INTERFACE PUBLIC LogCore EXTENDS __SYSTEM.IQueryInterface

// Logger method.
// Logs data in custom format. No additional formatting will be done.
METHOD LogCustomFormat : BOOL
VAR_INPUT
    data : Tc2_System.T_MaxString; // Data to be logged. No additional formatting will be done.
END_VAR
END_METHOD

// Logger method.
// Logs in the standard format. This includes
// - timestamp
// - log level
// - log message
// - instance path of logging source (optional)
// The message will only be logged if the logging level exceeds the configured minimum logging level.
METHOD LogStandardFormat : BOOL
VAR_INPUT
    data : Tc2_System.T_MaxString; // Data to be logged. Additional formatting wil be done.
    instance_path : Tc2_System.T_MaxString; // Instance path of calling logger to locate source of logging message.
    log_level : LogLevel; // Log level of message.
END_VAR
END_METHOD

// Logger method.
// Logs in standard format with additional structured key/value attributes.
// Backends that do not support structured attributes should forward data/instancePath/logLevel
// to their existing implementation and discard attrs/attr_count.
METHOD LogWithAttributes : BOOL
VAR_INPUT
    data : Tc2_System.T_MaxString;
    instance_path : Tc2_System.T_MaxString;
    log_level : LogLevel;
    attrs : ARRAY[0..9] OF LogAttribute;
    attr_count : USINT;
END_VAR
END_METHOD

END_INTERFACE

(* stored: Version 1.1.0.1
   Itf LogCore: Id {ed020564-7749-4641-89cc-c51a049d49ec}
   Method LogCustomFormat: Id {969f6a06-4b88-4def-b996-d34091c38c1e}
   Method LogStandardFormat: Id {445ed9e6-5cf6-4a42-b605-5d0ade9d322d}
   Method LogWithAttributes: Id {5ded2f7d-18a5-4fe2-9252-398da3dd842e} *)
